(* CODESYS project PackML_Example_RECOVERED_2024-11-19T12-11-37.project
   Title: PackML Example
   Version: 1.0.0.0
   Author: 3S - Smart Software Solutions GmbH
   Description: Example project for the PackML State Machine library.
   Company: 3S - Smart Software Solutions GmbH

Project tree, tasks and I/O mapping:
  Device : CODESYS Control Win V3 x64, CODESYS, version 3.5.20.0
    application PackMLUnitModeManager
      libraries: OMAC PackML State Machine, 1.0.0.4 (3S - Smart Software Solutions GmbH); Standard, 3.5.18.0 (System)
      task MainTask (cyclic, interval t#20ms, priority 1) calls PLC_PRG
      task VISU_TASK (cyclic, interval 100 ms, priority 31) calls VisuElems.Visu_Prg
      global variables GVL
      program PLC_PRG [ST]: SimulateActingStateComplete
      visualisation Visualization
    SoftMotion General Axis Pool : SoftMotion General Axis Pool, CODESYS, version 4.11.0.0
      Axis : SM_Drive_Virtual, 3S - Smart Software Solutions GmbH, order no. 1805, version 4.0.0.0
          settings: wDriveID = 3; iMovementType = 0; fSWMaxVelocity = 1e3; fSWMaxAcceleration = 1e5; fSWMaxDeceleration = 1e5
  Device2 : CODESYS Control Win V3 x64, CODESYS, version 3.5.20.0
    application PackMLAxisControl
      libraries: OMAC PackML State Machine, 1.0.0.4 (3S - Smart Software Solutions GmbH)
      task Task (cyclic, interval t#20ms, priority 1) calls PLC_PRG
      task VISU_TASK (cyclic, interval 100 ms, priority 31) calls VisuElems.Visu_Prg
      program PLC_PRG [ST]
      function block AxisControl [ST]
      image pool ImagePool
      visualisation Visualization
    SoftMotion General Axis Pool : SoftMotion General Axis Pool, CODESYS, version 4.11.0.0
      Axis : SM_Drive_Virtual, 3S - Smart Software Solutions GmbH, order no. 1805, version 4.0.0.0
          settings: wDriveID = 2; iMovementType = 0; fSWMaxVelocity = 1e3; fSWMaxAcceleration = 1e5; fSWMaxDeceleration = 1e5
  MyPackML : CODESYS Control Win V3 x64, CODESYS, version 3.5.20.0
    application Application
      libraries: OMAC PackML State Machine, 1.0.0.4 (3S - Smart Software Solutions GmbH); Standard, 3.5.18.0 (System)
      PackML/
        function block MyUnitMode [ST]
        function block FB_Generic [ST]: M_Clearing, M_Init, M_Complete, M_Suspended, ParseStateToString, M_Idle, M_Log, M_Held, M_Aborted, GenerateErrorMsg, M_Completing, M_Execute, M_Stopped, Callback, M_Unsuspending, M_Starting, M_Holding, M_Suspending, M_CheckError, M_Resetting, M_StateComplete, M_Aborting, M_Stopping, M_Unholding, M_mapping, M_Undefined
        PackML/
          State and Mode/
            data type E_PMLProtectedUnitMode
            data type ST_PMLSubUnitInfo
            data type E_PMLCommand
            data type E_PMLState
          data type ST_PMLStateMachineOptions
          global variables G_PML
          data type ST_PMLUnitModeConfiguration
          data type ST_ChangeIntoProduction
          ITFs/
            interface I_UnitState: M_Idle, M_Holding, M_Unholding, M_Stopped, M_Execute, M_Held, M_Starting, M_Complete, M_Aborted, M_Suspended, M_Clearing, M_Stopping, M_Reseting, M_StateComplete, M_Aborting, M_Undefined, M_Unsuspending, M_Suspending, M_Completing
            interface I_UnitStateActing: M_Unholding, M_Execute, M_Completing, M_Reseting, M_Starting, M_Holding, M_Suspending, M_Unsuspending, M_Clearing, M_StateComplete, M_Aborting, M_Stopping
            interface I_UnitStateWaiting: M_Held, M_Idle, M_Undefined, M_Stopped, M_Suspended, M_Aborted, M_Complete
          data type ST_PMLSubUnitInfoRef
          Machine State/
            function block PML_UnitModeConfig [ST]
            function block PML_StateMachine [ST]: _supportedStates, M_NextState, M_StateComplete
            function block PML_UnitModeManager [ST]: M_SwitchUnitMode, M_Register
          PackTags/
            data type ST_PackMLv30
            Common/
              data type ST_Product
              data type ST_Interface
              data type ST_Descriptor
              data type ST_EquipmentInterlock
              data type ST_Ingredient
              data type ST_Alarm
              data type ST_Count
            data type ST_PMLs
            data type ST_PMLc
            data type ST_PMLa
        PubSub/
          interface I_SubCallback: Callback
          interface I_PubSubService: Unsubscribe, Subscribe, Publish
          data type E_Topics
          data type PubSubData
          global variables G_PubSub
          function block PubSubService [ST]: Publish, Subscribe, Unsubscribe
          data type SubscriberCell
          data type KeyAndValue
        image pool ImagePool
        function block FB_Machine [ST]: M_Clearing, M_Starting, M_SetUnitInfo, M_Resetting
        function block FB_Sample [ST]: Callback, M_Completing, M_Resetting, ParseStateToString, M_Stopping, M_Holding, M_Starting, M_agingTest, M_Execute, M_Undefined, M_Idle, M_mapping, M_Aborting, M_Reset
        function block MyUnitModeManager [ST]
        DUTs/
          data type E_UnitName
          interface I_Common: M_Init, ParseStateToString, GenerateErrorMsg, M_Log
          data type ST_UnitInfo
          data type E_SampleStates
          data type E_PMLSupportState
          data type E_PMLUserUnitMode
          data type E_ServerityLevelType
        global variables GVL
  libraries: VisuSymbols, 4.5.0.0 (System)
  5ce3da45-db07-42e7-a21c-a00fff4ed8f6|C:\Users\a.werner\Documents\background.jpg
  5ce3da45-db07-42e7-a21c-a00fff4ed8f6|C:\Users\a.werner\Documents\background.jpg
  text list GlobalTextList
*)

// MyPackML/Application/PackML/PackML/State and Mode/E_PMLProtectedUnitMode
{attribute 'qualified_only'}
{attribute 'strict'}
TYPE E_PMLProtectedUnitMode :
(
	ePMLProtUnitMode_Invalid		:=	0,
	ePMLProtUnitMode_Production		:=	1,
	ePMLProtUnitMode_Maintenance	:= 	2,
	ePMLProtUnitMode_Manual	 		:=	3
);
END_TYPE

// MyPackML/Application/PackML/PackML/PackTags/ST_PackMLv30
TYPE ST_PackMLv30 :
STRUCT
	Command	: ST_PMLc;
	Status	: ST_PMLs;
	Admin	: ST_PMLa;
END_STRUCT
END_TYPE

// MyPackML/Application/PackML/PackML/ST_PMLStateMachineOptions
TYPE ST_PMLStateMachineOptions :
STRUCT
END_STRUCT
END_TYPE

// MyPackML/Application/PackML/PackML/PackTags/Common/ST_Product
TYPE ST_Product :
STRUCT
	 /// 
	 ///Product identification number 
	 ProductID: DINT; 
	 /// 
	 ///Parameters required for processing given product 
	 ProcessVariables: ARRAY[1..G_PML.MaxProductProcessVariables] OF ST_Descriptor; 
	 /// 
	 ///Ingredients required for processing given product 
	 Ingredients: ARRAY[1..G_PML.MaxIngredients] OF ST_Ingredient;	
END_STRUCT
END_TYPE

// MyPackML/Application/PackML/PackML/ST_PMLUnitModeConfiguration
TYPE ST_PMLUnitModeConfiguration :
	STRUCT
		bActive				: BOOL;				
		aStateDisabled		: ARRAY [E_PMLState.ePMLState_Undefined..E_PMLState.ePMLState_Complete] OF BOOL;				
		aModeChangeValid	: ARRAY [E_PMLState.ePMLState_Undefined..E_PMLState.ePMLState_Complete] OF BOOL;			
		sName				: STRING;
	END_STRUCT	
END_TYPE

// MyPackML/Application/PackML/PackML/ST_ChangeIntoProduction
//structure for a visu userwindow, to chnage into productionmode
TYPE ST_ChangeIntoProduction :
STRUCT
	bYes		: BOOL;
	bNo			: BOOL;
	bYesReset	: BOOL;
END_STRUCT
END_TYPE

// MyPackML/Application/PackML/DUTs/E_UnitName
//Enumeration for Machineunits
TYPE E_UnitName :
(
	eMachine		:= 1,
	eSample			:= 2
				
)DINT;
END_TYPE

// MyPackML/Application/PackML/PackML/PackTags/Common/ST_Interface
TYPE ST_Interface :
STRUCT
	 /// 
	 ///Identification number of upstream or downstream unit machine 
	 Number: DINT; 
	 /// 
	 ///Control command for upstream or downstream machine 
	 ControlCmdNumber: DINT; 
	 /// 
	 ///Control command value associated with ControlCmdNumber 
	 CmdValue: DINT; 
	 /// 
	 ///Parameter data required for peer-to-peer coordination 
	 Parameter: ARRAY[1..G_PML.MaxInterfaceParameters] OF ST_Descriptor;
END_STRUCT
END_TYPE

// MyPackML/Application/PackML/PackML/PackTags/Common/ST_Descriptor
TYPE ST_Descriptor :
STRUCT
	 /// 
	 ///Parameter identification number 
	 ID: DINT; 
	 /// 
	 ///Parameter description 
	 Name: STRING; 
	 /// 
	 ///Parameter units of measure 
	 Unit: STRING; 
	 /// 
	 ///Numeric value of parameter 
	 Value: REAL;
END_STRUCT
END_TYPE

// MyPackML/Application/PackML/DUTs/ST_UnitInfo
//structure includes unit information
TYPE ST_UnitInfo :
STRUCT
	Name		: STRING;
	ActState	: E_PMLState;
	ActMode		: DINT;
END_STRUCT
END_TYPE

// MyPackML/Application/PackML/PackML/PackTags/ST_PMLs
TYPE ST_PMLs :
STRUCT
	/// 
	///Numeric representation of the active unit mode (required) 
	UnitModeCurrent: DINT; 
	/// 
	///Handshaking bit acknowledging that unit mode change request has been made. 
	UnitModeRequested: BOOL; 
	/// 
	///Signals that unit mode change request has been accepted; switching is actively in process. 
	UnitModeChangeInProcess: BOOL; 
	/// 
	///Numeric representation of the active state (required) 
	StateCurrent: DINT; 
	/// 
	///Handshaking value acknowledging that state change request has been made. 
	StateRequested: DINT; 
	/// 
	///Signals that state change request has been accepted; switching is actively in process. 
	StateChangeInProcess: BOOL; 
	/// 
	///Active machine speed setpoint in units of [primary packages/min] (required) 
	MachSpeed: REAL; 
	/// 
	///Actual machine speed in units of [primary packages/min] (required) 
	CurMachSpeed: REAL; 
	/// 
	///Bitwise indication that materials are ready for processing. 
	MaterialInterlock: ARRAY[0..31] OF BOOL; 
	/// 
	///Signals that the machine is either blocked or starved (required) 
	EquipmentInterlock: ST_EquipmentInterlock; 
	/// 
	///Use to coordinate activities between peers (i.e. upstream or downstream unit machines.) 
	RemoteInterface: ARRAY [1..G_PML.MaxStatusRemoteInterfaces] OF ST_Interface; 
	/// 
	///Current values or parameters associated to the end user supervisory interface. 
	Parameter: ARRAY [1..G_PML.MaxStatusParameters] OF ST_Descriptor; 
	/// 
	///Current recipe or process data associated to the various products run on the unit machine. 
	Product: ARRAY [1..G_PML.MaxStatusProducts] OF ST_Product;	
END_STRUCT
END_TYPE

// MyPackML/Application/PackML/DUTs/E_SampleStates
{attribute 'qualified_only'}
{attribute 'strict'}
TYPE E_SampleStates :
(
	IDLE := 0,
	INIT,
	CHECK,
	WAIT,
	WAIT_ON,
	WAIT_OFF,
	DETECTION,
	LAMP_ON,
	LAMP_OFF,
	DONE,

	ERROR
);
END_TYPE

// MyPackML/Application/PackML/PackML/State and Mode/ST_PMLSubUnitInfo
TYPE ST_PMLSubUnitInfo :
STRUCT
	Active	: BOOL;				
	eState	: E_PMLState	:=	E_PMLState.ePMLState_Aborted;	
END_STRUCT
END_TYPE

// MyPackML/Application/PackML/PackML/PackTags/ST_PMLc
TYPE ST_PMLc :
STRUCT
	/// 
	///Numeric representation of the commanded unit mode (required) 
	UnitMode: DINT; 
	/// 
	///Signals request that the current value of Command.UnitMode be activated (required) 
	UnitModeChangeRequest: BOOL; 
	/// 
	///Machine speed setpoint in units of [primary packages/min] (required) 
	MachSpeed: REAL; 
	/// 
	///Bitwise indication that materials are ready for processing. 
	MaterialInterlock: ARRAY[1..32] OF BOOL; 
	/// 
	///Numerical representation of the state commands (1=Reset, 2=Start, etc.) (required) 
	CntrlCmd: DINT; 
	/// 
	///Signals request that the current value of Command.CntrlCmd be activated (required) 
	CmdChangeRequest: BOOL; 
	///
	///Use to coordinate activities between peers (i.e. upstream or downstream unit machines.) 
	RemoteInterface: ARRAY [1..G_PML.MaxCommandRemoteInterfaces] OF ST_Interface; 
	/// 
	///Values or parameters associated to the end user supervisory interface. 
	Parameter: ARRAY [1..G_PML.MaxCommandParameters] OF ST_Descriptor; 
	/// 
	///Recipe or process data associated to the various products run on the unit machine. 
	Product: ARRAY [1..G_PML.MaxCommandProducts] OF ST_Product;
	
END_STRUCT
END_TYPE

// MyPackML/Application/PackML/PubSub/E_Topics
TYPE E_Topics :
(
	UNKNOWN 				:= 0, 
	SAMPLE_SUBSCRRIBE_1		:= 1, 
	SAMPLE_SUBSCRRIBE_2		:= 2, 
	SAMPLE_SUBSCRRIBE_3		:= 3,
	NUMBER_OF_TOPICS
);
END_TYPE

// MyPackML/Application/PackML/PackML/ST_PMLSubUnitInfoRef
TYPE ST_PMLSubUnitInfoRef :
STRUCT
	//pArray			: PVOID;//codesys don't have pvoid yet	
	pArray			: POINTER TO ST_PMLSubUnitInfo;		
	ArraySize		: UDINT;				
	NoOfSubUnits	: UDINT;	
END_STRUCT
END_TYPE

// MyPackML/Application/PackML/PackML/PackTags/Common/ST_EquipmentInterlock
TYPE ST_EquipmentInterlock :
STRUCT
	/// 
	///Machine stoppage due to downstream fault 
	Blocked: BOOL; 
	/// 
	///Machine stoppage due to upstream or supply fault 
	Starved: BOOL;
END_STRUCT
END_TYPE

// MyPackML/Application/PackML/PubSub/PubSubData
TYPE PubSubData :
STRUCT
	Topic : E_Topics;
	Data	: ARRAY[0..MAX_PUB_SUB_DATA] OF KeyAndValue;
END_STRUCT
END_TYPE

// MyPackML/Application/PackML/PackML/PackTags/Common/ST_Ingredient
TYPE ST_Ingredient: 
STRUCT 
	 /// 
	 ///Ingredient identification number 
	 IngredientID: DINT; 
	 /// 
	 ///Parameters associated to given ingredient 
	 Parameter: ARRAY[1..G_PML.MaxIngredientParameters] OF ST_Descriptor; 
END_STRUCT 
END_TYPE

// MyPackML/Application/PackML/DUTs/E_PMLSupportState
{attribute 'qualified_only'}
{attribute 'strict'}
TYPE E_PMLSupportState :
(
	Stopped := 16#1, // Bit 0
	Resetting := 16#2, // Bit 1
	Idle := 16#4, // Bit 2
	Starting := 16#8, // Bit 3
	Execute := 16#10, // Bit 4
	Holding := 16#20, // Bit 5
	Held := 16#40, // Bit 6
	UnHolding := 16#80, // Bit 7
	Suspending := 16#100, // Bit 8
	Suspended := 16#200, // Bit 9
	UnSuspending := 16#400, // Bit 10
	Completing := 16#800, // Bit 11
	Complete := 16#1000, // Bit 12
	Stopping := 16#2000, // Bit 13
	Aborting := 16#4000, // Bit 14
	Aborted := 16#8000, // Bit 15
	Clearing := 16#10000, // Bit 16
	
	No := 0,
	All := 16#1FFFF,
	Invalid := 16#80000000
) DWORD;
END_TYPE

// MyPackML/Application/PackML/PackML/State and Mode/E_PMLCommand
{attribute 'strict'}
TYPE E_PMLCommand :
(
	ePMLCommand_Undefined		:=	0,	
	ePMLCommand_Reset			:=	1,	
	ePMLCommand_Start			:=	2,	
	ePMLCommand_Stop			:=	3,	
	ePMLCommand_Hold			:=	4,	
	ePMLCommand_Unhold			:=	5,	
	ePMLCommand_Suspend			:=	6,	
	ePMLCommand_Unsuspend		:=	7,	
	ePMLCommand_Abort			:=	8,	
	ePMLCommand_Clear			:=	9,	
	//	extension TO OMAC TR88.00.02
	ePMLCommand_Complete		:=	10
);
END_TYPE

// MyPackML/Application/PackML/PackML/PackTags/Common/ST_Alarm
TYPE ST_Alarm: 
STRUCT 
	 /// 
	 ///Alarm or warning current status 
	 Trigger: BOOL; 
	 /// 
	 ///Alarm or warning identification number 
	 ID: DINT; 
	 /// 
	 ///Context specific value associated to given alarm or warning 
	 Value: DINT; 
	 /// 
	 ///Alarm or warning description 
	 Message: STRING; 
	 /// 
	 ///Identification number associated to alarm type or severity 
	 Category: DINT; 
	 /// 
	 ///Time stamp of alarm or warning occurrence. Format year:month:day:hour:min:sec:µsec 
	 DateTime: ARRAY[0..6] OF DINT; 
	 /// 
	 ///Time stamp of alarm or warning acknowledgment. Format year:month:day:hour:min:sec:µsec 
	 AckDateTime: ARRAY[0..6] OF DINT; 
END_STRUCT 
END_TYPE

// MyPackML/Application/PackML/PackML/PackTags/Common/ST_Count
TYPE ST_Count :
STRUCT
	 /// 
	 ///Product identification number 
	 ID: DINT; 
	 /// 
	 ///Product description 
	 Name: STRING; 
	 /// 
	 ///Product unit of measure 
	 Unit: STRING; 
	 /// 
	 ///Count since last operator reset 
	 Count: DINT; 
	 /// 
	 ///Count since last accumulative counter reset 
	 AccCount: DINT;
END_STRUCT
END_TYPE

// MyPackML/Application/PackML/DUTs/E_PMLUserUnitMode
//Enumeration for User Modes
TYPE E_PMLUserUnitMode : (
	ePMLUnitMode_Service		:=  4,
	ePMLUnitMode_Usermode2		:=  5,
	ePMLUnitMode_Usermode3		:=  6,
	ePMLUnitMode_Usermode4		:=  7,
	ePMLUnitMode_Usermode5 		:=  8,
	ePMLUnitMode_Usermode6 		:=  9,
	ePMLUnitMode_Usermode7 		:=  10
) DINT;
END_TYPE

// MyPackML/Application/PackML/PubSub/SubscriberCell
TYPE SubscriberCell :
STRUCT
	occupied : BOOL;
	subscriber : I_SubCallback;
END_STRUCT
END_TYPE

// MyPackML/Application/PackML/PubSub/KeyAndValue
TYPE KeyAndValue :
STRUCT
	Key : STRING;
	Value : string;
END_STRUCT
END_TYPE

// MyPackML/Application/PackML/DUTs/E_ServerityLevelType
{attribute 'qualified_only'}
{attribute 'strict'}
TYPE E_ServerityLevelType :
(
	SERVICE := 0,
	ERROR,
	WARNING,
	INFO,
	DEBUG
);
END_TYPE

// MyPackML/Application/PackML/PackML/PackTags/ST_PMLa
TYPE ST_PMLa :
STRUCT
	/// 
	///Parameters associated to the local interface (e.g. HMI) 
	Parameter: ARRAY [1..G_PML.MaxAdminParameters] OF ST_Descriptor; 
	/// 
	///Listing of all currently active alarms 
	Alarm: ARRAY [1..G_PML.MaxAlarms] OF ST_Alarm; 
	/// 
	///Extent of the Alarm array 
	AlarmExtent: DINT	:= G_PML.MaxAlarms; 
	/// 
	///Chronological alarm history, with most recent given as AlarmHistory[0] 
	AlarmHistory: ARRAY [1..G_PML.MaxHistoryAlarms] OF ST_Alarm; 
	/// 
	///Extent of AlarmHistory array 
	AlarmHistoryExtent: DINT	:= G_PML.MaxHistoryAlarms; 
	/// 
	///Alarm associated to the primary cause of machine stoppage ('first fault') (required) 
	StopReason: ARRAY [1..G_PML.MaxStopReasons] OF ST_Alarm; 
	/// 
	///Extent of StopReason array 
	StopReasonExtent: DINT	:= G_PML.MaxStopReasons; 
	/// 
	///Listing of all currently active warnings 
	Warning: ARRAY [1..G_PML.MaxWarnings] OF ST_Alarm; 
	/// 
	///Extent of warning array 
	WarningExtent: DINT	:= G_PML.MaxWarnings; 
	/// 
	///Elapsed time in seconds of current mode. 
	ModeCurrentTime: ARRAY [0..G_PML.MaxUnitMode] OF DINT;
	/// 
	///Cumulative time in seconds in each defined mode. 
	ModeCumulativeTime: ARRAY [0..G_PML.MaxUnitMode] OF DINT; 
	/// 
	///Elapsed time in seconds of current [mode, state] pair. 
	StateCurrentTime: ARRAY [0..G_PML.MaxUnitMode, 0..G_PML.MaxMachineState] OF DINT; 
	/// 
	///Cumulative time in seconds in each defined [mode, state] pair. 
	StateCumulativeTime: ARRAY [0..G_PML.MaxUnitMode, 0..G_PML.MaxMachineState] OF DINT; 
	/// 
	///Count of raw materials used or consumed during production 
	ProdConsumedCount: ARRAY [1..G_PML.MaxConsumedCounts] OF ST_Count; 
	/// 
	///Count of total products (i.e. good + defective) made during production (required) 
	ProdProcessedCount: ARRAY [1..G_PML.MaxProductCounts] OF ST_Count; 
	/// 
 	///Count of defective products made during production. (required) 
	ProdDefectiveCount: ARRAY [1..G_PML.MaxProductCounts] OF ST_Count; 
	/// 
	///Accumulative time since last reset of timer arrays. 
	AccTimeSinceReset: DINT; 	
	/// 
	///Maximum design speed of the machine within given environment. 
	MachDesignSpeed: REAL; 	
	/// 
	///Bitwise indication of inactive states in current mode. 
	StatesDisabled: DINT; 		
	/// 
	///Current date and time of local processing unit (PLC, PC, PAC, microcontroller, etc.) 
	PLCDateTime: ARRAY[0..6] OF DINT;
END_STRUCT
END_TYPE

// MyPackML/Application/PackML/PackML/State and Mode/E_PMLState
TYPE E_PMLState :
(
	//states according TO PackTags v3.0
	ePMLState_Undefined		:=			0,	
	ePMLState_Clearing		:=			1,	
	ePMLState_Stopped		:=			2,	
	ePMLState_Starting		:=			3,	
	ePMLState_Idle			:=			4,	
	ePMLState_Suspended		:=			5,	
	ePMLState_Execute		:=			6,	
	ePMLState_Stopping		:=			7,	
	ePMLState_Aborting		:=			8,	
	ePMLState_Aborted		:=			9,	
	ePMLState_Holding		:=			10,	
	ePMLState_Held			:=			11,	
	ePMLState_Unholding		:=			12,	
	ePMLState_Suspending	:=			13,	
	ePMLState_Unsuspending	:=			14,	
	ePMLState_Resetting		:=			15,	
	ePMLState_Completing	:=			16,	
	ePMLState_Complete		:=			17
);
END_TYPE

// MyPackML/Application/PackML/PackML/G_PML
{attribute 'qualified_only'}
VAR_GLOBAL CONSTANT
	MaxInterfaceParameters		: INT	:=5;	//PMLc/PMLs
	MaxProductProcessVariables	: INT	:=10;
	MaxIngredients				: INT	:=10;
	MaxIngredientParameters		: INT	:=10;
	MaxCommandRemoteInterfaces	: INT	:=2;	//PMLc
	MaxCommandParameters		: INT	:=10;	
	MaxCommandProducts			: INT	:=5;
	MaxStatusRemoteInterfaces	: INT	:=2;	//PMLs
	MaxStatusParameters			: INT	:=10;	
	MaxStatusProducts			: INT	:=5;	
	MaxAdminParameters			: INT	:=10;	//PMLa
	MaxAlarms					: INT	:=10;	
	MaxHistoryAlarms			: INT	:=10;	
	MaxStopReasons				: INT	:=10;	
	MaxWarnings					: INT	:=10;	
	MaxConsumedCounts			: INT	:=10;	
	MaxProductCounts			: INT	:=10;
	
	MaxUnitMode					:INT	:=31;
	MaxMachineState				:INT	:=17;
	stPMLUnitModeConfiguration	:ARRAY [0..MaxUnitMode] OF ST_PMLUnitModeConfiguration	:=	[STRUCT(bActive := TRUE, sName := 'Invalid', aStateDisabled := [18(FALSE)], aModeChangeValid := [18(TRUE)]), 
																							 STRUCT(bActive := TRUE, sName := 'Production', aStateDisabled := [18(FALSE)], aModeChangeValid := [TRUE, FALSE, TRUE, FALSE, TRUE, FALSE, FALSE, FALSE, FALSE, TRUE, FALSE, TRUE, FALSE, FALSE, FALSE, FALSE, FALSE, FALSE]), 
																							 STRUCT(bActive := TRUE, sName := 'Maintenance', aStateDisabled := [FALSE, FALSE, FALSE, FALSE, FALSE, TRUE, FALSE, FALSE, FALSE, FALSE, FALSE, FALSE, FALSE, TRUE, TRUE, FALSE, TRUE, TRUE], aModeChangeValid := [TRUE, FALSE, TRUE, FALSE, TRUE, FALSE, FALSE, FALSE, FALSE, TRUE, FALSE, TRUE, FALSE, FALSE, FALSE, FALSE, FALSE, FALSE]), 
																							 STRUCT(bActive := TRUE, sName := 'Manual', aStateDisabled := [FALSE, FALSE, FALSE, FALSE, FALSE, TRUE, FALSE, FALSE, FALSE, FALSE, TRUE, TRUE, TRUE, TRUE, TRUE, FALSE, TRUE, TRUE], aModeChangeValid := [TRUE, FALSE, TRUE, FALSE, TRUE, FALSE, FALSE, FALSE, FALSE, TRUE, FALSE, FALSE, FALSE, FALSE, FALSE, FALSE, FALSE, FALSE])];	
END_VAR

// Device/PackMLUnitModeManager/GVL
VAR_GLOBAL CONSTANT
	gc_sPRODUCTION 	: STRING := 'Production';
	gc_sSEMIAUTO 	: STRING := 'Semi Auto';
	gc_sSETUP 		: STRING := 'Setup';
	gc_sUSER		: STRING := 'User';
END_VAR

// MyPackML/Application/PackML/PubSub/G_PubSub

VAR_GLOBAL CONSTANT
	MAX_PUB_SUB_DATA	: INT:=19;
END_VAR

// MyPackML/Application/PackML/GVL
VAR_GLOBAL CONSTANT
	gc_sPRODUCTION : STRING := 'Production';
	gc_sSEMIAUTO : STRING := 'Semi Auto';
	gc_sSETUP : STRING := 'Setup';
END_VAR
{attribute 'qualified_only'}
VAR_GLOBAL
	packTags	: ST_PackMLv30;
	bButtonProductionReq		: BOOL;							//TRUE when a mode change to PRODUCTION is requested
	stChangeIntoProduction		: ST_ChangeIntoProduction;		//Result of command box "Change to Production requested"
	
	PubSubService	: PubSubService;

	pml_adminAlarm	: PML_AdminAlarm;
	
	aUnitInfo					: ARRAY [1..12] OF ST_UnitInfo;	//Array includes the states and modes of machineunits	
	aCaption					: ARRAY [1..12] OF STRING := ['F1','F2','F3','F4','F5','F6','F7','F8','F9','F10','F11','F12'];
	aKeyPressed					: ARRAY [1..12] OF BOOL;


	fb_sample	: FB_Sample;		
END_VAR

// Device2/PackMLAxisControl/PLC_PRG
PROGRAM PLC_PRG
VAR
	xInit				: BOOL := FALSE; // Flag for initialization

	ac: AxisControl;
	
	// Visu Commands	
	xAbort				: BOOL;
	xActingStateComplete: BOOL;
	xClear				: BOOL;
	xHold				: BOOL;
	xReset				: BOOL;
	xStart				: BOOL;
	xStop				: BOOL;
	xSuspend			: BOOL;
	xUnHold				: BOOL;
	xUnSuspend			: BOOL;
	
	
END_VAR

ac(Axis:=Axis);

// Visu commands
IF xAbort THEN
	ac.ItfUnitMode.Abort();
END_IF
IF xClear THEN
	ac.ItfUnitMode.Clear();
END_IF
IF xHold THEN
	ac.ItfUnitMode.Hold();
END_IF
IF xReset THEN
	ac.ItfUnitMode.Reset();
END_IF
IF xStart THEN
	ac.ItfUnitMode.Start();
END_IF
IF xStop THEN
	ac.ItfUnitMode.Stop();
END_IF
IF xSuspend THEN
	ac.ItfUnitMode.Suspend();
END_IF
IF xUnHold THEN
	ac.ItfUnitMode.UnHold();
END_IF
IF xUnSuspend THEN
	ac.ItfUnitMode.UnSuspend();
END_IF
IF xActingStateComplete AND ac.ItfUnitMode.CurrentState = PACK_ML.State.Execute THEN
	ac.ItfUnitMode.ActingStateCompleted();
END_IF

END_PROGRAM

// Device/PackMLUnitModeManager/PLC_PRG
// Example project for the PackML State Machine with three unit modes.
PROGRAM PLC_PRG
VAR
	productionUnitMode	: PACK_ML.UnitMode; // Example unit mode for prodction
	semiAutoUnitMode	: PACK_ML.UnitMode; // Example unit mode for semi auto production
	setupUnitMode		: PACK_ML.UnitMode; // Example unit mode for setup
	userUnitMode		: PACK_ML.UnitMode; // Example unit mode for setup
	unitModeManager		: PACK_ML.UnitModeManager; // Unit mode manager to switch between unitmodes
	currentUnitMode		: PACK_ML.IUnitMode;
	xInit				: BOOL := FALSE; // Flag for initialization
	
	// Visu Commands	
	xAbort				: BOOL;
	xActingStateComplete: BOOL;
	xClear				: BOOL;
	xHold				: BOOL;
	xReset				: BOOL;
	xStart				: BOOL;
	xStop				: BOOL;
	xSuspend			: BOOL;
	xUnHold				: BOOL;
	xUnSuspend			: BOOL;
	
	// Helper
	xSimulate			: BOOL;
	xChangeState		: BOOL := FALSE;	
	timer1				: TON;	
	iSelectedUnitMode	: INT := 0;
	iLastSelectedUnitMode: INT := 0;
	xUserModeChanged	: BOOL;
	
END_VAR

IF NOT xInit THEN
	productionUnitMode(		sName := gc_sPRODUCTION, 
							dwSupportedStates := PACK_ML.State.All, 
							dwAllowsLeavingFromStates := PACK_ML.State.Stopped OR PACK_ML.State.Aborted OR PACK_ML.State.Idle, 
							dwAllowsEnteringIntoStates := PACK_ML.State.Stopped OR PACK_ML.State.Aborted OR PACK_ML.State.Idle, 
							eInitialState := PACK_ML.State.Idle,
							xActive := TRUE);
	semiAutoUnitMode(		sName := gc_sSEMIAUTO, 
							dwSupportedStates := PACK_ML.State.All - PACK_ML.State.Completing - PACK_ML.State.Complete - PACK_ML.State.Holding - PACK_ML.State.Held - PACK_ML.State.UnHolding,
							dwAllowsLeavingFromStates := PACK_ML.State.Stopped OR PACK_ML.State.Aborted OR PACK_ML.State.Idle, 
							dwAllowsEnteringIntoStates := PACK_ML.State.Stopped OR PACK_ML.State.Aborted OR PACK_ML.State.Idle,   
							eInitialState := PACK_ML.State.Idle, 
							xActive := FALSE);
	setupUnitMode(			sName := gc_sSETUP, 
							dwSupportedStates := PACK_ML.State.All - PACK_ML.State.Completing - PACK_ML.State.Complete - PACK_ML.State.Holding - PACK_ML.State.Held - PACK_ML.State.UnHolding - PACK_ML.State.UnSuspending - PACK_ML.State.Suspended - PACK_ML.State.Suspending,
							dwAllowsLeavingFromStates := PACK_ML.State.Stopped OR PACK_ML.State.Aborted OR PACK_ML.State.Idle,   
							dwAllowsEnteringIntoStates := PACK_ML.State.Stopped OR PACK_ML.State.Aborted OR PACK_ML.State.Idle, 
							eInitialState := PACK_ML.State.Idle, 
							xActive := FALSE);
	userUnitMode(			sName := gc_sUSER, 
							dwSupportedStates := PACK_ML.State.All - PACK_ML.State.Completing - PACK_ML.State.Complete - PACK_ML.State.Holding - PACK_ML.State.Held - PACK_ML.State.UnHolding - PACK_ML.State.UnSuspending - PACK_ML.State.Suspended - PACK_ML.State.Suspending-PACK_ML.State.Clearing-PACK_ML.Aborted,
							dwAllowsLeavingFromStates := PACK_ML.State.Stopped OR PACK_ML.State.Aborted OR PACK_ML.State.Idle,   
							dwAllowsEnteringIntoStates := PACK_ML.State.Stopped OR PACK_ML.State.Aborted OR PACK_ML.State.Idle, 
							eInitialState := PACK_ML.State.Idle, 
							xActive := FALSE);
	// Register the unit modes 
	unitModeManager.Register(productionUnitMode);
	unitModeManager.Register(semiAutoUnitMode);
	unitModeManager.Register(setupUnitMode);
	unitModeManager.Register(userUnitMode);
	xInit := TRUE;
END_IF

IF unitModeManager.ActiveUnitMode <> 0 THEN	
	currentUnitMode := unitModeManager.ActiveUnitMode;
	
	// Visu commands
	IF xAbort THEN
		unitModeManager.ActiveUnitMode.Abort();
	END_IF
	IF xClear THEN
		unitModeManager.ActiveUnitMode.Clear();
	END_IF
	IF xHold THEN
		unitModeManager.ActiveUnitMode.Hold();
	END_IF
	IF xReset THEN
		unitModeManager.ActiveUnitMode.Reset();
	END_IF
	IF xStart THEN
		unitModeManager.ActiveUnitMode.Start();
	END_IF
	IF xStop THEN
		unitModeManager.ActiveUnitMode.Stop();
	END_IF
	IF xSuspend THEN
		unitModeManager.ActiveUnitMode.Suspend();
	END_IF
	IF xUnHold THEN
		unitModeManager.ActiveUnitMode.UnHold();
	END_IF
	IF xUnSuspend THEN
		unitModeManager.ActiveUnitMode.UnSuspend();
	END_IF
	IF xActingStateComplete AND NOT xSimulate THEN
		unitModeManager.ActiveUnitMode.ActingStateCompleted();
	END_IF
	
	// Simulate action complete
	SimulateActingStateComplete();	 
END_IF

// Change the current unit mode
IF iSelectedUnitMode <> iLastSelectedUnitMode THEN
	CASE iSelectedUnitMode OF 
		0:
			xUserModeChanged := unitModeManager.SwitchUnitMode(gc_sPRODUCTION);
		1:
			xUserModeChanged := unitModeManager.SwitchUnitMode(gc_sSEMIAUTO);
		2:
			xUserModeChanged := unitModeManager.SwitchUnitMode(gc_sSETUP);
		3:
			xUserModeChanged := unitModeManager.SwitchUnitMode(gc_sUser);
	END_CASE
	IF xUserModeChanged THEN
		iLastSelectedUnitMode := iSelectedUnitMode;
	ELSE
		iSelectedUnitMode := iLastSelectedUnitMode;
	END_IF
END_IF

METHOD SimulateActingStateComplete
VAR_INPUT
END_VAR
VAR
	nextSupportedState	: UDINT;	
END_VAR
nextSupportedState := unitModeManager.ActiveUnitMode.NextState(unitModeManager.ActiveUnitMode.CurrentState);	
IF nextSupportedState = PACK_ML.State.Execute OR nextSupportedState = PACK_ML.State.Completing OR nextSupportedState = PACK_ML.State.Complete OR nextSupportedState = PACK_ML.State.Held OR nextSupportedState = PACK_ML.State.Aborted OR nextSupportedState = PACK_ML.State.Stopped OR nextSupportedState = PACK_ML.State.Idle OR nextSupportedState = PACK_ML.State.Suspended THEN	
	timer1(IN := TRUE, PT := T#2S, Q => xChangeState);
	xSimulate := TRUE;
END_IF   
IF xChangeState THEN
	unitModeManager.ActiveUnitMode.ActingStateCompleted();
	timer1(IN := FALSE);
	xSimulate := FALSE;
	xChangeState := FALSE;
END_IF
END_METHOD

END_PROGRAM

// Device2/PackMLAxisControl/AxisControl
FUNCTION_BLOCK AxisControl
// This FB represents an axis, which is controlled according to its active unit mode
VAR_IN_OUT
	Axis: AXIS_REF_SM3;
END_VAR
VAR_OUTPUT
	ItfUnitMode	: PACK_ML.IUnitMode; // UnitMode of the axis
END_VAR
VAR
	UM	: PACK_ML.UnitMode; 

	xInit				: BOOL := FALSE; // Flag for initialization

	//motion FBs
	p: MC_Power;
	rs: MC_ReadStatus;
	res: MC_Reset;
	moverel: MC_MoveRelative;
	halt: MC_Halt;
	moveabs: MC_MoveAbsolute;
	h: MC_Home;
	
	
	tii	: TON;
END_VAR

IF NOT xInit THEN	
	UM				(		sName := 'Normal Operation', 
							dwSupportedStates := PACK_ML.State.All - PACK_ML.State.Suspending - PACK_ML.State.Suspended - PACK_ML.State.UnSuspending, 
							dwAllowsLeavingFromStates := PACK_ML.State.Stopped OR PACK_ML.State.Aborted OR PACK_ML.State.Idle, 
							dwAllowsEnteringIntoStates := PACK_ML.State.Stopped OR PACK_ML.State.Aborted OR PACK_ML.State.Idle, 
							eInitialState := PACK_ML.State.Aborted,
							xActive := TRUE);
	ItfUnitMode := UM; 
	xInit := TRUE;
END_IF

CASE UM.CurrentState OF
PACK_ML.State.Stopped,
PACK_ML.State.Aborted,
PACK_ML.State.Idle,
PACK_ML.State.Held,
PACK_ML.State.Complete :
	// in this waiting states we reset the Execute input of the moving FBs
	res.Execute := FALSE;
	moverel.Execute := FALSE;
	halt.Execute := FALSE;
	moveabs.Execute := FALSE;
	h.Execute := FALSE;
PACK_ML.State.Resetting :
	IF rs.Errorstop THEN	//first reset errors when necessary
		h.Execute := FALSE;
		IF res.Error THEN
			res.Execute := FALSE;
		ELSE	
			res.Execute := TRUE;
		END_IF
	ELSE
		p.bDriveStart := TRUE;	//release quickstop
		IF p.Status THEN
			h.Execute := TRUE;	//do homing
			IF h.Done THEN	
				h.Execute := FALSE;
				UM.ActingStateCompleted();
			END_IF
		END_IF
	END_IF
PACK_ML.State.Starting :
	moverel.Execute:=FALSE;
	UM.ActingStateCompleted();
PACK_ML.State.Execute :
	moverel.Execute:=TRUE;
	IF moverel.Done THEN
		moverel.Execute:=FALSE;
 	END_IF
PACK_ML.State.Holding :
	moverel.Execute:=FALSE;
	halt.Execute:=TRUE;
	IF halt.Done THEN
		halt.Execute := FALSE;
		UM.ActingStateCompleted();
	END_IF
PACK_ML.State.UnHolding :
	halt.Execute:=FALSE;
	moveabs.Execute := TRUE;
	IF moveabs.Done THEN
		moveabs.Execute := FALSE;
		UM.ActingStateCompleted();
	END_IF
PACK_ML.State.Completing :
	IF moverel.Done THEN
		UM.ActingStateCompleted();
	END_IF
PACK_ML.State.Aborting :
	p.bDriveStart := FALSE;
	p.bRegulatorOn := FALSE;
	UM.ActingStateCompleted();
PACK_ML.State.Stopping,
PACK_ML.State.Clearing :	
	p.bRegulatorOn:=TRUE; 
	p.bDriveStart:=FALSE; 
	IF p.bRegulatorRealState AND NOT p.bDriveStartRealState THEN
		UM.ActingStateCompleted();
	END_IF
END_CASE

p(
	Axis:=Axis , 
	Enable:=TRUE , 
	Status=> , 
	bRegulatorRealState=> , 
	bDriveStartRealState=> , 
	Busy=> , 
	Error=> , 
	ErrorID=> );

rs(
	Axis:=Axis , 
	Enable:=TRUE , 
	Valid=> , 
	Busy=> , 
	Error=> , 
	ErrorID=> , 
	Disabled=> , 
	Errorstop=> , 
	Stopping=> , 
	StandStill=> , 
	DiscreteMotion=> , 
	ContinuousMotion=> , 
	SynchronizedMotion=> , 
	Homing=> , 
	ConstantVelocity=> , 
	Accelerating=> , 
	Decelerating=> , 
	FBErrorOccured=> );
	
res(
	Axis:=Axis , 
	Execute:= , 
	Done=> , 
	Busy=> , 
	Error=> , 
	ErrorID=> );
	
moverel(
	Axis:=Axis , 
	Distance:=360 , 
	Velocity:=360 , 
	Acceleration:=360 , 
	Deceleration:=360, 
	Jerk:= , 
	Done=> , 
	Busy=> , 
	CommandAborted=> , 
	Error=> , 
	ErrorID=> );
	
moveabs(
	Axis:=Axis , 
	Execute:= , 
	Position:=0 , 
	Velocity:=360 , 
	Acceleration:=360 , 
	Deceleration:=360 , 
	Jerk:= , 
	Direction:=positive , 
	Done=> , 
	Busy=> , 
	CommandAborted=> , 
	Error=> , 
	ErrorID=> );
	
halt(
	Axis:=axis , 
	Execute:= , 
	Deceleration:=1000 , 
	Jerk:= , 
	Done=> , 
	Busy=> , 
	CommandAborted=> , 
	Error=> , 
	ErrorID=> );
	
h(
	Axis:=Axis , 
	Execute:= , 
	Position:= , 
	Done=> , 
	Busy=> , 
	CommandAborted=> , 
	Error=> , 
	ErrorID=> );

END_FUNCTION_BLOCK

// MyPackML/Application/PackML/PubSub/I_SubCallback
(*
Description: 
Interface that every function block that wants to be a subscriber, needs to implement.
*)
INTERFACE I_SubCallback

(*
Description: 
the callback that will be invoked when there is a publish for what the subscriber was subscribed to.
*)
METHOD Callback
VAR_INPUT
	data : PubSubData;
END_VAR
END_METHOD

END_INTERFACE

// MyPackML/Application/PackML/PackML/Machine State/PML_UnitModeConfig
//just to config the unit mode,can 
FUNCTION_BLOCK PML_UnitModeConfig
VAR_INPUT
	//
	eMode							: DINT;				
	sName							: STRING;
	//config which state disable				
	bDisableClearing				: BOOL;				
	bDisableStarting				: BOOL;				
	bDisableSuspended				: BOOL;				
	bDisableStopping				: BOOL;				
	bDisableAborting				: BOOL;				
	bDisableHolding					: BOOL;				
	bDisableHeld					: BOOL;				
	bDisableUnholding				: BOOL;				
	bDisableSuspending				: BOOL;				
	bDisableUnsuspending			: BOOL;				
	bDisableResetting				: BOOL;				
	bDisableIdle					: BOOL;				
	bDisableCompleting				: BOOL;				
	bDisableComplete				: BOOL;
	//config unit mode can be changed in which state				
	bEnableUnitModeChangeStopped	: BOOL;				
	bEnableUnitModeChangeIdle		: BOOL;				
	bEnableUnitModeChangeSuspended	: BOOL;				
	bEnableUnitModeChangeExecute	: BOOL;				
	bEnableUnitModeChangeAborted	: BOOL;				
	bEnableUnitModeChangeHeld		: BOOL;				
	bEnableUnitModeChangeComplete	: BOOL;		
END_VAR
VAR_OUTPUT
	bError	: BOOL;				
	nErrorId	: UDINT;	
END_VAR
VAR
END_VAR

END_FUNCTION_BLOCK

// MyPackML/Application/PackML/MyUnitMode
FUNCTION_BLOCK MyUnitMode
VAR_INPUT
END_VAR
VAR_OUTPUT
END_VAR
VAR
END_VAR

END_FUNCTION_BLOCK

// MyPackML/Application/PackML/PackML/ITFs/I_UnitState
INTERFACE I_UnitState EXTENDS I_UnitStateWaiting,I_UnitStateActing

METHOD M_Idle
VAR_INPUT
END_VAR
END_METHOD

METHOD M_Holding
VAR_INPUT
END_VAR
END_METHOD

METHOD M_Unholding
VAR_INPUT
END_VAR
END_METHOD

METHOD M_Stopped
VAR_INPUT
END_VAR
END_METHOD

METHOD M_Execute
VAR_INPUT
END_VAR
END_METHOD

METHOD M_Held
VAR_INPUT
END_VAR
END_METHOD

METHOD M_Starting
VAR_INPUT
END_VAR
END_METHOD

METHOD M_Complete
VAR_INPUT
END_VAR
END_METHOD

METHOD M_Aborted
VAR_INPUT
END_VAR
END_METHOD

METHOD M_Suspended
VAR_INPUT
END_VAR
END_METHOD

METHOD M_Clearing
VAR_INPUT
END_VAR
END_METHOD

METHOD M_Stopping
VAR_INPUT
END_VAR
END_METHOD

METHOD M_Reseting
VAR_INPUT
END_VAR
END_METHOD

METHOD M_StateComplete
VAR_INPUT
END_VAR
END_METHOD

METHOD M_Aborting
VAR_INPUT
END_VAR
END_METHOD

METHOD M_Undefined
VAR_INPUT
END_VAR
END_METHOD

METHOD M_Unsuspending
VAR_INPUT
END_VAR
END_METHOD

METHOD M_Suspending
VAR_INPUT
END_VAR
END_METHOD

METHOD M_Completing
VAR_INPUT
END_VAR
END_METHOD

END_INTERFACE

// MyPackML/Application/PackML/PackML/ITFs/I_UnitStateWaiting
INTERFACE I_UnitStateWaiting

METHOD M_Held
VAR_INPUT
END_VAR
END_METHOD

METHOD M_Idle
VAR_INPUT
END_VAR
END_METHOD

METHOD M_Undefined
VAR_INPUT
END_VAR
END_METHOD

METHOD M_Stopped
VAR_INPUT
END_VAR
END_METHOD

METHOD M_Suspended
VAR_INPUT
END_VAR
END_METHOD

METHOD M_Aborted
VAR_INPUT
END_VAR
END_METHOD

METHOD M_Complete
VAR_INPUT
END_VAR
END_METHOD

END_INTERFACE

// MyPackML/Application/PackML/PackML/ITFs/I_UnitStateActing
INTERFACE I_UnitStateActing

METHOD M_Unholding
VAR_INPUT
END_VAR
END_METHOD

METHOD M_Execute
VAR_INPUT
END_VAR
END_METHOD

METHOD M_Completing
VAR_INPUT
END_VAR
END_METHOD

METHOD M_Reseting
VAR_INPUT
END_VAR
END_METHOD

METHOD M_Starting
VAR_INPUT
END_VAR
END_METHOD

METHOD M_Holding
VAR_INPUT
END_VAR
END_METHOD

METHOD M_Suspending
VAR_INPUT
END_VAR
END_METHOD

METHOD M_Unsuspending
VAR_INPUT
END_VAR
END_METHOD

METHOD M_Clearing
VAR_INPUT
END_VAR
END_METHOD

METHOD M_StateComplete
VAR_INPUT
END_VAR
END_METHOD

METHOD M_Aborting
VAR_INPUT
END_VAR
END_METHOD

METHOD M_Stopping
VAR_INPUT
END_VAR
END_METHOD

END_INTERFACE

// MyPackML/Application/PackML/DUTs/I_Common
INTERFACE I_Common

METHOD M_Init : BOOL
VAR_INPUT
END_VAR
END_METHOD

METHOD ParseStateToString : STRING
VAR_INPUT
END_VAR
END_METHOD

METHOD GenerateErrorMsg : STRING
VAR_INPUT
	errorType	: STRING;
//	strState	: STRING;
	iState		: INT;
	errorMsg	: STRING;
END_VAR
END_METHOD

METHOD M_Log : STRING
VAR_INPUT
	eLogType	: E_ServerityLevelType;
	sTextLog	: STRING;
END_VAR
END_METHOD

END_INTERFACE

// MyPackML/Application/PackML/PackML/Machine State/PML_StateMachine
//can be bypass the state which is disable according to the configuration of eMode
//example:if disable clearing and resetting,when it command=clear/reset it will bybass M_Clearing and M_Stopped
//output estate according to eCommand ,then the subunit call the corresponding method according to the estate
FUNCTION_BLOCK PML_StateMachine
VAR_INPUT
	eMode				: DINT	:= E_PMLProtectedUnitMode.ePMLProtUnitMode_Production;
	eCommand			: E_PMLCommand;			
	stSubUnitInfoRef	: ST_PMLSubUnitInfoRef;	//determing machine's state according to the subUnits		
	stOptions			: ST_PMLStateMachineOptions;		
END_VAR
VAR_OUTPUT
	eState		:E_PMLState	:= ePMLState_Undefined;
	sState		:STRING;		
	bError		:BOOL;	
	nErrorID	:UDINT;	
END_VAR
VAR
	eCurrentState	: E_PMLState	:= ePMLState_Undefined;
	dwSupportedStates : DWORD := 2#11111111111111111; // Supported states
	bInit: BOOL;
END_VAR

PROPERTY _supportedStates : DWORD
GET
_supportedStates	:= dwSupportedStates;
END_GET
SET
END_SET
END_PROPERTY

// Get the next machine state without checking the supported states.
//todo:get the next machine state with checking the supported states
METHOD M_NextState : E_PMLState
VAR_INPUT
	e : E_PMLState;
END_VAR
CASE e OF
ePMLState_Stopped:
	M_NextState := ePMLState_Resetting;
ePMLState_Resetting:
	M_NextState := ePMLState_Idle;
ePMLState_Idle:
	M_NextState := ePMLState_Starting;
ePMLState_Starting:
	M_NextState := ePMLState_Execute;
ePMLState_Execute://
	M_NextState := ePMLState_Undefined;
ePMLState_Holding:
	M_NextState := ePMLState_Held;
ePMLState_Held:
	M_NextState := ePMLState_Unholding;
ePMLState_Unholding:
	M_NextState := ePMLState_Execute;
ePMLState_Suspending:
	M_NextState := ePMLState_Suspended;
ePMLState_Suspended:
	M_NextState := ePMLState_Unsuspending;
ePMLState_Unsuspending:
	M_NextState := ePMLState_Execute;
ePMLState_Completing:
	M_NextState := ePMLState_Complete;
ePMLState_Complete:
	M_NextState := ePMLState_Resetting;
ePMLState_Stopping:	
	M_NextState := ePMLState_Stopped;
ePMLState_Aborting:
	M_NextState := ePMLState_Aborted;
ePMLState_Aborted:
	M_NextState := ePMLState_Clearing;
ePMLState_Clearing:
	M_NextState := ePMLState_Stopped;
END_CASE
END_METHOD

// This method should be called by the program if an action has been finished.
//if not 
METHOD M_StateComplete : BOOL
VAR_INPUT
END_VAR
CASE eState OF
	ePMLState_Undefined:
		M_StateComplete	:= FALSE;
	ePMLState_Clearing:
		IF (TO_DWORD(M_NextState(eState)) AND _supportedStates) = 0 THEN//disable clearing
			M_StateComplete := FALSE;
			RETURN;
		END_IF	
		eState := M_NextState(eState);
		M_StateComplete := TRUE;
	ePMLState_Starting:
	//
	ePMLState_Stopping:	
	//
	ePMLState_Aborting:
	//
	ePMLState_Holding:
	//
	ePMLState_Unholding:
	//
	ePMLState_Suspending:
	//
	ePMLState_Unsuspending:
	//
	ePMLState_Resetting:
	//
	ePMLState_Completing:
	//
	
	
	
	ePMLState_Complete:
	//
	ePMLState_Stopped:
	//	
	ePMLState_Idle:
	//
	ePMLState_Suspended:
	//
	ePMLState_Execute:
	//
	ePMLState_Aborted:
	//
	ePMLState_Held:
	//
END_CASE
END_METHOD

END_FUNCTION_BLOCK

// MyPackML/Application/PackML/FB_Generic
//the functionblock FB_Generick is transmitted to every machineunit
FUNCTION_BLOCK FB_Generic IMPLEMENTS I_UnitState,I_SubCallback,I_Common
VAR_INPUT
	eModeCommand			: DINT;									//Mode from superior Unit
	eCommand				: E_PMLCommand := ePMLCommand_Abort;	//Command for a new state from superior unit
END_VAR
VAR_OUTPUT
	eMode					: DINT;									//Actual mode of the Unit
	eState					: E_PMLState (*:= ePMLState_Aborted*) ;	//Actual state of the Unit
	
	bUndefinedDone			: BOOL;									//When the SPS is started, the first state is Undefiend. bUndefined is TRUE, when the method Undefined has succesful finished
	bInvalidModeCommandOut	: BOOL;
	bChangeIntoProduction	: BOOL;
END_VAR
VAR
	fbUnitModeManager		: PML_UnitModeManager;					//The PML_UnitModeManager manage the Modechanges
	fbStateMachine 			: PML_StateMachine;						//The PML_StateMachine mangae the Statechanges
	
	nStateModeChange		: INT	:= 0;							//Variable to handle the modechange
	nLastState				: E_PMLState;							//Variable to store last state
	
	packTags				: ST_PackMLv30;
	i	: INT;
	
	ton_timeout			: TON;
	iStateTemp			: INT;	
	
	rTrig_electricalError	:ARRAY[0..10] OF R_TRIG;
	alarm_temp		: ST_Alarm;
	subscribed	: BOOL	:= FALSE;
	subData		: PubSubData;
	
	strState	: STRING;
	sComponent_name			: STRING;
	iComponetID				: INT;	
	infoLevel	: E_ServerityLevelType;//should be set to high level after debug
END_VAR

M_mapping();
CASE nStateModeChange OF
0:
	//Waiting for user request
	bChangeIntoProduction:= FALSE;
	IF  GVL.bButtonProductionReq AND (GVL.PackTags.Command.UnitMode = ePMLProtUnitMode_Production) AND (GVL.PackTags.Status.UnitModeCurrent = ePMLProtUnitMode_Invalid) THEN
			nStateModeChange	:= 1;
	ELSIF  GVL.PackTags.Command.UnitModeChangeRequest AND (GVL.PackTags.Command.UnitMode <> ePMLProtUnitMode_Production) THEN
			nStateModeChange	:= 1;
	ELSIF  GVL.bButtonProductionReq AND (GVL.PackTags.Command.UnitMode = ePMLProtUnitMode_Production) AND (GVL.PackTags.Status.UnitModeCurrent <> ePMLProtUnitMode_Production) THEN
			nStateModeChange	:= 3;
	END_IF
1:
	//Starting UnitModeManager 
	fbUnitModeManager.bExecute				:= TRUE;
	fbUnitModeManager.eModeCommand			:= eModeCommand;
	GVL.PackTags.Status.UnitModeChangeInProcess	:= TRUE;

	IF fbUnitModeManager.bDone THEN
		fbUnitModeManager.bExecute	:= FALSE;
		bInvalidModeCommandOut		:= FALSE;
		nStateModeChange			:= 0;
		bChangeIntoProduction		:= FALSE;
		GVL.PackTags.Status.UnitModeChangeInProcess	:= FALSE;
	ELSIF fbUnitModeManager.bError THEN
		bInvalidModeCommandOut		:= TRUE;
		fbUnitModeManager.bExecute	:= FALSE;
		nLastState					:= GVL.packTags.Status.StateCurrent;
		nStateModeChange			:= 2;
		bChangeIntoProduction		:= FALSE;
		GVL.PackTags.Status.UnitModeChangeInProcess	:= FALSE;
	END_IF
2:
	//ErrorHanddling
	IF  GVL.PackTags.Command.UnitModeChangeRequest THEN
		nStateModeChange:=0;
		bInvalidModeCommandOut		:= FALSE;
	ELSIF nLastState<> GVL.PackTags.Status.StateCurrent THEN
		bInvalidModeCommandOut		:= FALSE;
	END_IF
	
3:
	//state to check, if command 'Porduction' is valid
	IF (GVL.PackTags.Status.StateCurrent = ePMLState_Aborted OR GVL.PackTags.Status.StateCurrent = ePMLState_Stopped OR GVL.PackTags.Status.StateCurrent = ePMLState_Idle) THEN
		bChangeIntoProduction		:= TRUE;
		IF  GVL.stChangeIntoProduction.bYes OR GVL.stChangeIntoProduction.bYesReset THEN
			nStateModeChange			:= 1;		
		ELSIF GVL.stChangeIntoProduction.bNo THEN
			nStateModeChange			:= 0;
		END_IF
	ELSE
		nStateModeChange:= 2;
		bInvalidModeCommandOut		:= TRUE;
		nLastState					:= GVL.PackTags.Status.StateCurrent;
	END_IF
END_CASE


fbUnitModeManager(									
	eState			:= eState,
	eModeStatus		=> eMode,
	bDone			=> ,
	bError			=> ,
	nErrorId		=> );


IF fbUnitModeManager.eModeStatus <>  0 THEN
	//Calling the StateMachine, when there is a valid Mode
	fbStateMachine(
		eMode				:= eMode, 				
		eCommand			:= eCommand,			
		stSubUnitInfoRef	:= ,
		stOptions			:= , 
		eState				=> eState, 				
		bError				=> , 
		nErrorID			=> );
END_IF

//One of the methods is executing  by the actual state
CASE eState OF
	ePMLState_Undefined:
		M_Undefined();
	ePMLState_Clearing:
		M_Clearing();
	ePMLState_Stopped:
		M_Stopped();
	ePMLState_Starting:
		M_Starting();
	ePMLState_Idle:
		M_Idle();
	ePMLState_Suspended:
		M_Suspended();
	ePMLState_Execute:
		M_Execute();
	ePMLState_Stopping:
		M_Stopping();
	ePMLState_Aborting:
		M_Aborting();
	ePMLState_Aborted:
		M_Aborted();
	ePMLState_Holding:
		M_Holding();
	ePMLState_Held:
		M_Held();
	ePMLState_Unholding:
		M_Unholding();
	ePMLState_Suspending:
		M_Suspending();
	ePMLState_Unsuspending:
		M_Unsuspending();
	ePMLState_Resetting:
		M_Resetting();
	ePMLState_Completing:
		M_Completing();
	ePMLState_Complete:
		M_Complete();
END_CASE

{attribute 'object_name' := 'M_Clearing'}
METHOD M_Clearing
M_StateComplete();
END_METHOD

METHOD M_Init : BOOL
VAR_INPUT
END_VAR
END_METHOD

{attribute 'object_name' := 'M_Complete'}
METHOD M_Complete
END_METHOD

{attribute 'object_name' := 'M_Suspended'}
METHOD M_Suspended
END_METHOD

METHOD ParseStateToString : STRING
VAR_INPUT
END_VAR
END_METHOD

{attribute 'object_name' := 'M_Idle'}
METHOD M_Idle
END_METHOD

(*
M_Log method :
*)
METHOD M_Log : STRING
VAR_INPUT
	eLogType	: E_ServerityLevelType;
	sTextLog	: STRING;	
END_VAR
IF eLogType <= infoLevel THEN
//
END_IF
END_METHOD

{attribute 'object_name' := 'M_Held'}
METHOD M_Held
END_METHOD

{attribute 'object_name' := 'M_Aborted'}
METHOD M_Aborted
END_METHOD

(*
GenerateErrorMsg method:generate the error message according to the inputs
generate example:'{M9906} fb_sample DETECTION time out for T#3s.'
errorType:
		'M':mechanical error
		'E':electrical error
		'S':safety error
iState:state of state machine
errorMsg:descirbe the error
sComponent_name:defined in every componet
iComponetID:defined in every componet
strState:parseStateToString() to get the strState in ervery component
sTimeout_setting:defined in every componet
*)
METHOD GenerateErrorMsg : STRING
VAR_INPUT
	errorType	: STRING;
	iState		: INT;
	errorMsg	: STRING;	
END_VAR
VAR
	errorID	: INT;
END_VAR
GenerateErrorMsg	:= '';
GenerateErrorMsg	:= CONCAT('{',errorType);
IF iComponetID<10 THEN
	errorID	:= iComponetID*1000+iState;
ELSE
	errorID	:= iComponetID*100+iState;
END_IF
GenerateErrorMsg	:= CONCAT(GenerateErrorMsg,INT_TO_STRING(errorID));
GenerateErrorMsg	:= CONCAT(GenerateErrorMsg,'} ');
GenerateErrorMsg	:= CONCAT(GenerateErrorMsg,sComponent_name);
GenerateErrorMsg	:= CONCAT(GenerateErrorMsg,' ');
GenerateErrorMsg	:= CONCAT(GenerateErrorMsg,strState);
GenerateErrorMsg	:= CONCAT(GenerateErrorMsg,' ');
GenerateErrorMsg	:= CONCAT(GenerateErrorMsg,errorMsg);
IF errorMsg='time out' THEN
	GenerateErrorMsg	:= CONCAT(GenerateErrorMsg,' ');
	GenerateErrorMsg	:= CONCAT(GenerateErrorMsg,'for ');
	GenerateErrorMsg	:= CONCAT(GenerateErrorMsg,TIME_TO_STRING(ton_timeout.PT));//timeout setting
	GenerateErrorMsg	:= CONCAT(GenerateErrorMsg,'.');
END_IF
END_METHOD

{attribute 'object_name' := 'M_Completing'}
METHOD M_Completing
M_StateComplete();
END_METHOD

{attribute 'object_name' := 'M_Execute'}
METHOD M_Execute

M_StateComplete();
END_METHOD

{attribute 'object_name' := 'M_Stopped'}
METHOD M_Stopped
END_METHOD

(*
Description: 
the callback that will be invoked when there is a publish for what the subscriber was subscribed to.
*)
METHOD Callback
VAR_INPUT
	data : PubSubData;
END_VAR
END_METHOD

{attribute 'object_name' := 'M_Unsuspending'}
METHOD M_Unsuspending
VAR_INPUT
END_VAR
M_StateComplete();
END_METHOD

{attribute 'object_name' := 'M_Starting'}
METHOD M_Starting
M_StateComplete();
END_METHOD

{attribute 'object_name' := 'M_Holding'}
METHOD M_Holding
M_StateComplete();
END_METHOD

{attribute 'object_name' := 'M_Suspending'}
METHOD M_Suspending
VAR_INPUT
END_VAR
M_StateComplete();
END_METHOD

METHOD M_CheckError : BOOL
VAR_INPUT
END_VAR

VAR
	Trigger: INT;
END_VAR
M_CheckError	:= FALSE;

FOR i:=1 TO G_PML.MaxAlarms DO
	IF THIS^.PackTags.Admin.Alarm[i].Trigger THEN
		M_CheckError	:= TRUE;
	END_IF
END_FOR
END_METHOD

{attribute 'object_name' := 'M_Resetting'}
METHOD M_Resetting
M_StateComplete();
END_METHOD

{attribute 'object_name' := 'M_StateComplete'}
METHOD M_StateComplete
//the actual state is completed
fbStateMachine.M_StateComplete();
END_METHOD

{attribute 'object_name' := 'M_Aborting'}
METHOD M_Aborting
M_StateComplete();
END_METHOD

{attribute 'object_name' := 'M_Stopping'}
METHOD M_Stopping
M_StateComplete();
END_METHOD

{attribute 'object_name' := 'M_Unholding'}
METHOD M_Unholding
VAR_INPUT
END_VAR
M_StateComplete();
END_METHOD

METHOD M_mapping : BOOL
VAR_INPUT
END_VAR
alarm_temp.DateTime	:=GVL.packTags.Admin.PlcDateTime;
END_METHOD

{attribute 'object_name' := 'M_Undefined'}
METHOD M_Undefined
END_METHOD

END_FUNCTION_BLOCK

// MyPackML/Application/PackML/PackML/Machine State/PML_UnitModeManager
//if estate is enable to switch mode
FUNCTION_BLOCK PML_UnitModeManager
VAR_INPUT
	bExecute		: BOOL;				
	eModeCommand	: DINT;				
	eState			: E_PMLState;	//for decide if mode can be change,if can,change and done,if not,error with errorid	
END_VAR
VAR_OUTPUT
	eModeStatus	: DINT;				
	sModeStatus	: STRING;				
	bDone		: BOOL;				
	bError		: BOOL;				
	nErrorId	: UDINT;
END_VAR
VAR
END_VAR

// Switch to an other unit mode and check the permission.
// Returns true if switching is allowed, returns false if switching is forbidden.
METHOD M_SwitchUnitMode : BOOL
VAR_INPUT
	sModeName: STRING; // Name of the unit mode to switch
END_VAR
END_METHOD

// Registers an unit mode
METHOD M_Register : BOOL
VAR_INPUT
	
END_VAR
END_METHOD

END_FUNCTION_BLOCK

// MyPackML/Application/PackML/FB_Sample
FUNCTION_BLOCK FB_Sample EXTENDS FB_Generic
VAR_INPUT
END_VAR
VAR_OUTPUT
END_VAR
VAR
	lamp			: BOOL;	
	eStates			: E_SampleStates := E_SampleStates.IDLE;;
	eStateTemp		: E_SampleStates := E_SampleStates.IDLE;
	
END_VAR

SUPER^();
IF NOT subscribed THEN
	GVL.PubSubService.Subscribe(E_Topics.SAMPLE_SUBSCRRIBE_1,THIS^);
	GVL.PubSubService.Subscribe(E_Topics.SAMPLE_SUBSCRRIBE_2,THIS^);
	GVL.PubSubService.Subscribe(E_Topics.SAMPLE_SUBSCRRIBE_3,THIS^);
END_IF
subscribed	:= TRUE;


sComponent_name		:= 'fb_sample';
iComponetID			:= 99;
strState	:= ParseStateToString();
infoLevel	:= E_ServerityLevelType.WARNING;

(*
Description: 
the callback that will be invoked when there is a publish for what the subscriber was subscribed to.
*)
METHOD Callback
VAR_INPUT
	data : PubSubData;
END_VAR
CASE data.Topic OF
	E_Topics.SAMPLE_SUBSCRRIBE_1:
		//ADSLOGSTR(msgCtrlMask:= ADSLOG_MSGTYPE_LOG,msgFmtStr:='get data from publish 1',strArg:='');
	E_Topics.SAMPLE_SUBSCRRIBE_2:
		//ADSLOGSTR(msgCtrlMask:= ADSLOG_MSGTYPE_LOG,msgFmtStr:='get data from publish 2',strArg:='');
	E_Topics.SAMPLE_SUBSCRRIBE_3:
		//ADSLOGSTR(msgCtrlMask:= ADSLOG_MSGTYPE_LOG,msgFmtStr:='get data from publish 3',strArg:='');		
END_CASE
END_METHOD

{attribute 'object_name' := 'M_Completing'}
METHOD M_Completing
CASE fbUnitModeManager.eModeStatus OF
	ePMLProtUnitMode_Production:
		;
END_CASE
END_METHOD

{attribute 'object_name' := 'M_Resetting'}
METHOD M_Resetting
CASE fbUnitModeManager.eModeStatus OF
	ePMLProtUnitMode_Production:		//Production, Mantainance, Manual
		lamp	:= FALSE;
		eStates :=E_SampleStates.IDLE;
		M_StateComplete();
	
	ePMLProtUnitMode_Maintenance, ePMLProtUnitMode_Manual, ePMLUnitMode_Service:
		M_StateComplete();
END_CASE
END_METHOD

METHOD ParseStateToString : STRING
VAR_INPUT
END_VAR
CASE THIS^.eStates OF
	E_SampleStates.IDLE:
		ParseStateToString	:='IDLE';
	E_SampleStates.INIT:
		ParseStateToString	:='INIT';
	E_SampleStates.CHECK:
		ParseStateToString	:='CHECK';
	E_SampleStates.DETECTION:	
		ParseStateToString	:='DETECTION';
	E_SampleStates.LAMP_ON:
		ParseStateToString	:='LAMP_ON';
	E_SampleStates.LAMP_OFF:
		ParseStateToString	:='LAMP_OFF';
	E_SampleStates.WAIT:
		ParseStateToString	:='WAIT';
	E_SampleStates.WAIT_ON:
		ParseStateToString	:='WAIT_ON';
	E_SampleStates.WAIT_OFF:
		ParseStateToString	:='WAIT_OFF';
	E_SampleStates.DONE:	
		ParseStateToString	:='DONE';
	E_SampleStates.ERROR:
		ParseStateToString	:='ERROR';
	ELSE
		ParseStateToString	:='UNKNOW STATE';
END_CASE
END_METHOD

{attribute 'object_name' := 'M_Stopping'}
METHOD M_Stopping
CASE fbUnitModeManager.eModeStatus OF
	ePMLProtUnitMode_Production, ePMLProtUnitMode_Manual:
				//////////////////////////////////////////////////////////timeout//////////////////////////////////////////	
		iStateTemp	:= eStateTemp;
		ton_timeout();
		IF eStateTemp=eStates THEN
			ton_timeout.IN	:=TRUE;
		ELSE
			ton_timeout.IN	:=FALSE;
			eStateTemp	:= eStates;	
		END_IF
		IF ton_timeout.Q THEN	
			ton_timeout.IN	:=FALSE;
			CASE eStates OF		
				E_SampleStates.IDLE:						
					;
				E_SampleStates.INIT:
					;
				E_SampleStates.WAIT_ON:
					;
				E_SampleStates.WAIT_OFF:
					;			
				E_SampleStates.ERROR:	
					alarm_temp.Message	:= 'Sample in error state';
				ELSE
					alarm_temp.Message	:= 'UNKNOWN STATES in Sample module';
			END_CASE
			IF eStates<>E_SampleStates.IDLE AND eStates<>E_SampleStates.WAIT_ON AND eStates<>E_SampleStates.WAIT_OFF THEN
				GVL.pml_adminAlarm.M_SetAlarm(stAdmin:=GVL.PackTags.Admin,stAlarm:=alarm_temp);
			END_IF
		END_IF
		
		CASE eStates OF 
				E_SampleStates.IDLE:						
					eStates	:= E_SampleStates.INIT;				
				E_SampleStates.INIT:
					ton_timeout.PT	:= T#1S;
					eStates	:= E_SampleStates.WAIT_ON; 
				E_SampleStates.WAIT_ON:
					lamp	:= TRUE;
					IF ton_timeout.Q THEN
						eStates	:= E_SampleStates.WAIT_OFF;
					END_IF
				E_SampleStates.WAIT_OFF:
					lamp	:= FALSE;
					IF ton_timeout.Q THEN
						eStates	:= E_SampleStates.IDLE;
						M_StateComplete();	
					END_IF
				E_SampleStates.ERROR:
					;
			END_CASE			
	ePMLProtUnitMode_Maintenance, ePMLUnitMode_Service:
		M_StateComplete();	
			//not defined
END_CASE
END_METHOD

{attribute 'object_name' := 'M_Holding'}
METHOD M_Holding
CASE fbUnitModeManager.eModeStatus OF
	ePMLProtUnitMode_Production:		//Mode Production
		//Finisch the actual seperationstep	
		

	ePMLProtUnitMode_Maintenance:
		M_StateComplete();
END_CASE
END_METHOD

{attribute 'object_name' := 'M_Starting'}
METHOD M_Starting
CASE fbUnitModeManager.eModeStatus OF
	ePMLProtUnitMode_Production:		//Production, Mantainance, Manual
		
		M_StateComplete();
	ePMLProtUnitMode_Maintenance, ePMLProtUnitMode_Manual, ePMLUnitMode_Service:
		M_StateComplete();
END_CASE
END_METHOD

METHOD M_agingTest : BOOL
VAR_INPUT
	
END_VAR
END_METHOD

{attribute 'object_name' := 'M_Execute'}
METHOD M_Execute

CASE fbUnitModeManager.eModeStatus OF
	ePMLProtUnitMode_Production:		//Mode Production
		//////////////////////////////////////////////////////////timeout//////////////////////////////////////////	
		iStateTemp	:= eStateTemp;
		ton_timeout();
		IF eStateTemp=eStates THEN
			ton_timeout.IN	:=TRUE;
		ELSE
			ton_timeout.IN	:=FALSE;
			eStateTemp	:= eStates;	
			M_Log(eLogType:=E_ServerityLevelType.INFO,sTextLog:='');
			IF ton_timeout.Q THEN
				RETURN;
			END_IF
		END_IF
		IF ton_timeout.Q THEN	
			ton_timeout.IN	:=FALSE;
			CASE eStates OF	
				E_SampleStates.ERROR:	
					alarm_temp.Message	:= GenerateErrorMsg(errorType:='M',iState := iStateTemp,errorMsg:='in error state.');
				ELSE
				alarm_temp.Message	:= GenerateErrorMsg(errorType:='M',iState := iStateTemp,errorMsg:='time out');
			END_CASE
			
//			CASE eStates OF		
//				E_SampleStates.IDLE:						
//					;
//				E_SampleStates.INIT:
//					;
//				E_SampleStates.WAIT_ON:
//					;
//				E_SampleStates.WAIT_OFF:
//					;			
//				E_SampleStates.ERROR:	
//					alarm_temp.Message	:= 'Sample in error state';
//				ELSE
//					alarm_temp.Message	:= 'UNKNOWN STATES in Sample module';
//			END_CASE
			IF eStates<>E_SampleStates.IDLE AND eStates<>E_SampleStates.WAIT_ON AND eStates<>E_SampleStates.WAIT_OFF THEN
				GVL.pml_adminAlarm.M_SetAlarm(stAdmin:=GVL.PackTags.Admin,stAlarm:=alarm_temp);
			END_IF
		END_IF
		
		CASE eStates OF 
				E_SampleStates.IDLE:
					ton_timeout.PT	:= T#1MS;						
					eStates	:= E_SampleStates.INIT;				
				E_SampleStates.INIT:
					ton_timeout.PT	:= T#1S;
					eStates	:= E_SampleStates.WAIT_ON; 
				E_SampleStates.DETECTION:
					ton_timeout.PT	:= T#3S;
				E_SampleStates.WAIT:
					ton_timeout.PT	:= T#200MS;					
				E_SampleStates.WAIT_ON:
					lamp	:= TRUE;
					IF ton_timeout.Q THEN
						eStates	:= E_SampleStates.WAIT_OFF;
					END_IF
				E_SampleStates.WAIT_OFF:
					lamp	:= FALSE;
					IF ton_timeout.Q THEN
						eStates	:= E_SampleStates.IDLE;
					END_IF
				E_SampleStates.ERROR:
					;
			END_CASE
		
		
	ePMLProtUnitMode_Maintenance, ePMLUnitMode_Service:		
		//
		
	ePMLProtUnitMode_Manual:		//Manaul

END_CASE
END_METHOD

{attribute 'object_name' := 'M_Undefined'}
METHOD M_Undefined

bUndefinedDone					:= TRUE;
END_METHOD

{attribute 'object_name' := 'M_Idle'}
METHOD M_Idle
// IF G_HMI.bAging_test THEN
// 	//M_agingTest();
// END_IF
END_METHOD

METHOD M_mapping : BOOL
VAR_INPUT
END_VAR
END_METHOD

{attribute 'object_name' := 'M_Aborting'}
METHOD M_Aborting
CASE fbUnitModeManager.eModeStatus OF	
	ePMLProtUnitMode_Production, ePMLProtUnitMode_Manual:		
		lamp	:= FALSE;		
		M_StateComplete();
			
	ePMLProtUnitMode_Maintenance, ePMLUnitMode_Service:
		
		M_StateComplete();
END_CASE
END_METHOD

METHOD M_Reset
VAR_INPUT
END_VAR
//Take away all commands
IF GVL.stChangeIntoProduction.bYesReset THEN
;
END_IF
END_METHOD

END_FUNCTION_BLOCK

// MyPackML/Application/PackML/PubSub/PubSubService
FUNCTION_BLOCK PubSubService IMPLEMENTS I_PubSubService
VAR_INPUT
END_VAR
VAR_OUTPUT
END_VAR

VAR
	TopicsToSubscribers : ARRAY[0..MAX_TOPICS - 1, 0..MAX_SUBSCRIBERS_PER_TOPIC - 1] OF SubscriberCell;
	subscriberCounters : ARRAY [0..MAX_TOPICS - 1] OF INT;
END_VAR

VAR CONSTANT 
	MAX_SUBSCRIBERS_PER_TOPIC : INT := 20;
	{attribute 'analysis' := '-33'}
	MAX_TOPICS : INT := E_Topics.NUMBER_OF_TOPICS;
END_VAR

METHOD Publish
VAR_INPUT
	topic	: E_Topics;
	data	: PubSubData;
END_VAR
VAR
	index : INT;
END_VAR
FOR index := 0 TO MAX_SUBSCRIBERS_PER_TOPIC -1 BY 1 DO
	IF TopicsToSubscribers[topic, index].OCCUPIED = TRUE THEN
		TopicsToSubscribers[topic, index].subscriber.Callback(data);
	END_IF
END_FOR
END_METHOD

METHOD Subscribe : INT
VAR_INPUT
	topic	: E_Topics;
	subCallback	: I_SubCallback;
END_VAR
VAR 
	index : INT;
END_VAR
Subscribe := -1;

IF  subscriberCounters[topic] >= MAX_SUBSCRIBERS_PER_TOPIC THEN
	RETURN;
END_IF

FOR index := 0 TO (MAX_SUBSCRIBERS_PER_TOPIC - 1) BY 1 DO
	IF TopicsToSubscribers[topic, index].occupied = FALSE THEN
		TopicsToSubscribers[topic, index].occupied := TRUE;
		TopicsToSubscribers[topic, index].subscriber := subCallback;
		Subscribe := index;
		subscriberCounters[topic] := subscriberCounters[topic] + 1;
		RETURN;
	END_IF
END_FOR
END_METHOD

METHOD Unsubscribe
VAR_INPUT
	topic : E_Topics;
	subscriberID	: INT;
END_VAR
IF TopicsToSubscribers[topic, subscriberID].occupied = TRUE THEN
	TopicsToSubscribers[topic, subscriberID].occupied := FALSE;
	subscriberCounters[topic] := subscriberCounters[topic] - 1; 	
END_IF
END_METHOD

END_FUNCTION_BLOCK

// MyPackML/Application/PackML/PubSub/I_PubSubService
(*
Description:
An interface to form the contract for a basic Publisher/Subscriber service.
explaination for each method is located at the method's place.
*)
INTERFACE I_PubSubService

(*
Description:
Through this method you can unsubcribe to a topic you've already subscribed beforehand.

Params: topic - the type of topic you wish to unsubscribe to
Params: subscriberID - the ID you've received from the subscribe method.
*)
METHOD Unsubscribe
VAR_INPUT
	topic : E_Topics;
	subscriberID : INT;
END_VAR
END_METHOD

(*
Description:
Through this method you can subcribe to a topic and be notified via the I_SubCallback interface.

Params: topic - the type of topic you wish to subscribe to
Params: subCallback - is a reference to subscribe who needs to implement the O_SubCallback interface.
Return: INT - this is an ID you need to keep in order to be able to use the Unsubscribe method.
		ID > 0 is a valid ID, ID = -1 meaning the you've failed to subscribe.
*)
METHOD Subscribe : INT
VAR_INPUT
	topic : E_Topics;
	subCallback :  I_SubCallback;
END_VAR
END_METHOD

(*
Description:
Through this method you can publish data to a certain topic domain

Params: topic - the type of topic you wish to publish data to.
Params: data - the data you wish to send to said topic.
*)
METHOD Publish
VAR_INPUT
	topic : E_Topics;
	data  : PubSubData;
END_VAR
END_METHOD

END_INTERFACE

// MyPackML/Application/PackML/FB_Machine
FUNCTION_BLOCK FB_Machine EXTENDS FB_Generic
VAR_INPUT

END_VAR
VAR_OUTPUT

END_VAR
VAR	

	
	stSubModuleInfo		: ARRAY [1..iSubModule] OF ST_PMLSubUnitInfo;	//Informations about the Subunits


	
	
END_VAR
VAR CONSTANT
	iSubModule	: UDINT :=1;
END_VAR

GVL.fb_sample(
	eModeCommand:= eModeCommand, 
	eCommand:= eCommand, 
	eMode=> , 
	eState=> stSubModuleInfo[iSubModule].eState, 
	bUndefinedDone=> , 
	bInvalidModeCommandOut=> , 
	bChangeIntoProduction=> );
stSubModuleInfo[iSubModule].Active		:= TRUE;

IF  GVL.fb_sample.bUndefinedDone  THEN
	bUndefinedDone := TRUE;
END_IF

//The fbStateMachine from FB_Machine gets the Information about the states and activity from the subunits
fbStateMachine.stSubUnitInfoRef.ArraySize		:= SIZEOF(stSubModuleInfo);
fbStateMachine.stSubUnitInfoRef.NoOfSubUnits	:= iSubModule;
fbStateMachine.stSubUnitInfoRef.pArray			:= ADR(stSubModuleInfo);



//Set unit information 
M_SetUnitInfo();


SUPER^();

{attribute 'object_name' := 'M_Clearing'}
METHOD M_Clearing

CASE fbUnitModeManager.eModeStatus OF
	ePMLProtUnitMode_Production:		//Production, Mantainance, Manual
		FOR i:=1 TO MaxAlarms DO
			GVL.pml_adminAlarm.M_AcknowledgeAlarm(stAdmin:=GVL.PackTags.Admin,stAlarm:=GVL.PackTags.Admin.Alarm[i]);
			GVL.pml_adminAlarm.M_ClearAlarm(stAdmin:=GVL.PackTags.Admin,stAlarm:=GVL.PackTags.Admin.Alarm[i]);
		END_FOR	
		M_StateComplete();		
// 		IF MAIN.application.safety.M_reset() THEN
// 			IF MAIN.application.safety.xError THEN
// 				eCommand	:= ePMLCommand_Abort;
// 			ELSE
// 				M_StateComplete();
// 			END_IF
// 		END_IF	
		
	
	ePMLProtUnitMode_Maintenance, ePMLProtUnitMode_Manual, ePMLUnitMode_Service:
		M_StateComplete();
END_CASE
END_METHOD

{attribute 'object_name' := 'M_Starting'}
METHOD M_Starting
CASE fbUnitModeManager.eModeStatus OF
	ePMLProtUnitMode_Production:		//Production, Mantainance, Manual
		//Resetting all Commands and Value
// 		G_HMI.bAging_test	:= FALSE;
		M_StateComplete();
	ePMLProtUnitMode_Maintenance, ePMLProtUnitMode_Manual, ePMLUnitMode_Service:
		M_StateComplete();
END_CASE
END_METHOD

METHOD M_SetUnitInfo
VAR_INPUT
END_VAR
GVL.aUnitInfo[eMachine].Name			:= 'fbMachine';
GVL.aUnitInfo[eMachine].ActMode			:= eMode;
GVL.aUnitInfo[eMachine].ActState		:= eState;

GVL.aUnitInfo[eSample].Name				:= 'fb_sample';
GVL.aUnitInfo[eSample].ActMode			:= GVL.fb_sample.eMode;
GVL.aUnitInfo[eSample].ActState			:= GVL.fb_sample.eState;
END_METHOD

{attribute 'object_name' := 'M_Resetting'}
METHOD M_Resetting
CASE fbUnitModeManager.eModeStatus OF
	ePMLProtUnitMode_Production:		//Production, Mantainance, Manual	
// 		IF MAIN.application.safety.M_reset() THEN
// 			IF MAIN.application.safety.xError THEN
// 				eCommand	:= ePMLCommand_Abort;
// 			ELSE
// 				M_StateComplete();
// 			END_IF
// 		END_IF	
		M_StateComplete();
	
	ePMLProtUnitMode_Maintenance, ePMLProtUnitMode_Manual, ePMLUnitMode_Service:
		M_StateComplete();
END_CASE
END_METHOD

END_FUNCTION_BLOCK

// MyPackML/Application/PackML/MyUnitModeManager
FUNCTION_BLOCK MyUnitModeManager
VAR_INPUT
END_VAR
VAR_OUTPUT
END_VAR
VAR
END_VAR

END_FUNCTION_BLOCK

// Device/PackMLUnitModeManager/Visualization
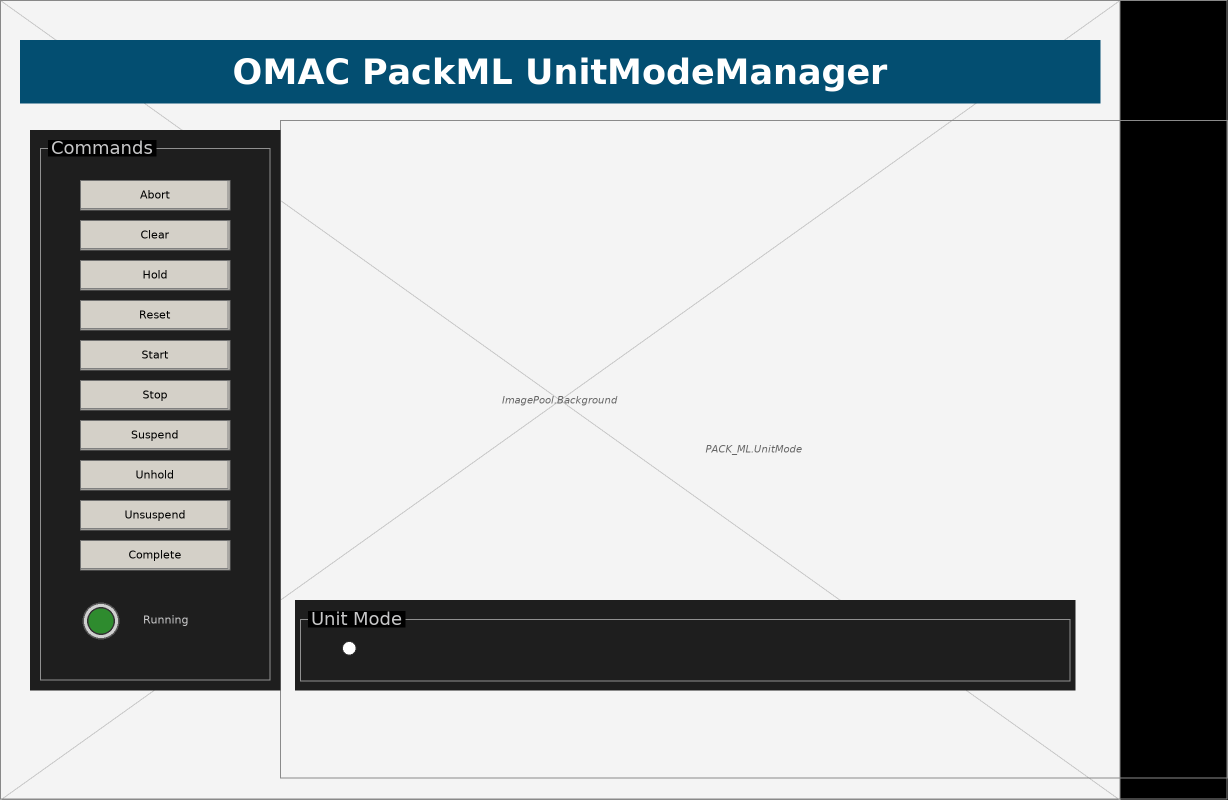
VISUALIZATION Visualization  // 1228x800
    Image (0,0 1120x800), image: ImagePool.Background
    Frame (280,120 948x658)
        shows PACK_ML.UnitMode(um := PLC_PRG.currentUnitMode)
    Rectangle (295,600 780x90)
    Rectangle (30,130 250x560)
    GroupBox (40,140 230x540), "Commands"
        Lamp1 (40,460 42x42), variable: PLC_PRG.xSimulate, style: Lamp-Lamp1-Green
        Label (100,465 57x30), "Running"
        Button (40,40 150x30), "Abort"
            tap PLC_PRG.xAbort
        Button (40,80 150x30), "Clear"
            tap PLC_PRG.xClear
        Button (40,120 150x30), "Hold"
            tap PLC_PRG.xHold
        Button (40,160 150x30), "Reset"
            tap PLC_PRG.xReset
        Button (40,200 150x30), "Start"
            tap PLC_PRG.xStart
        Button (40,240 150x30), "Stop"
            tap PLC_PRG.xStop
        Button (40,280 150x30), "Suspend"
            tap PLC_PRG.xSuspend
        Button (40,320 150x30), "Unhold"
            tap PLC_PRG.xUnHold
        Button (40,360 150x30), "Unsuspend"
            tap PLC_PRG.xUnSuspend
        Button (40,400 150x30), "Complete"
            tap PLC_PRG.xActingStateComplete
    GroupBox (300,611 770x70), "Unit Mode"
        RadioButton (40,20 700x34), variable: PLC_PRG.iSelectedUnitMode
            Areas[0]: Text=Production
            Areas[1]: Text=Semi Auto Production
            Areas[2]: Text=Setup
    Rectangle (20,40 1080x63), "OMAC PackML UnitModeManager"
END_VISUALIZATION

// Device2/PackMLAxisControl/Visualization
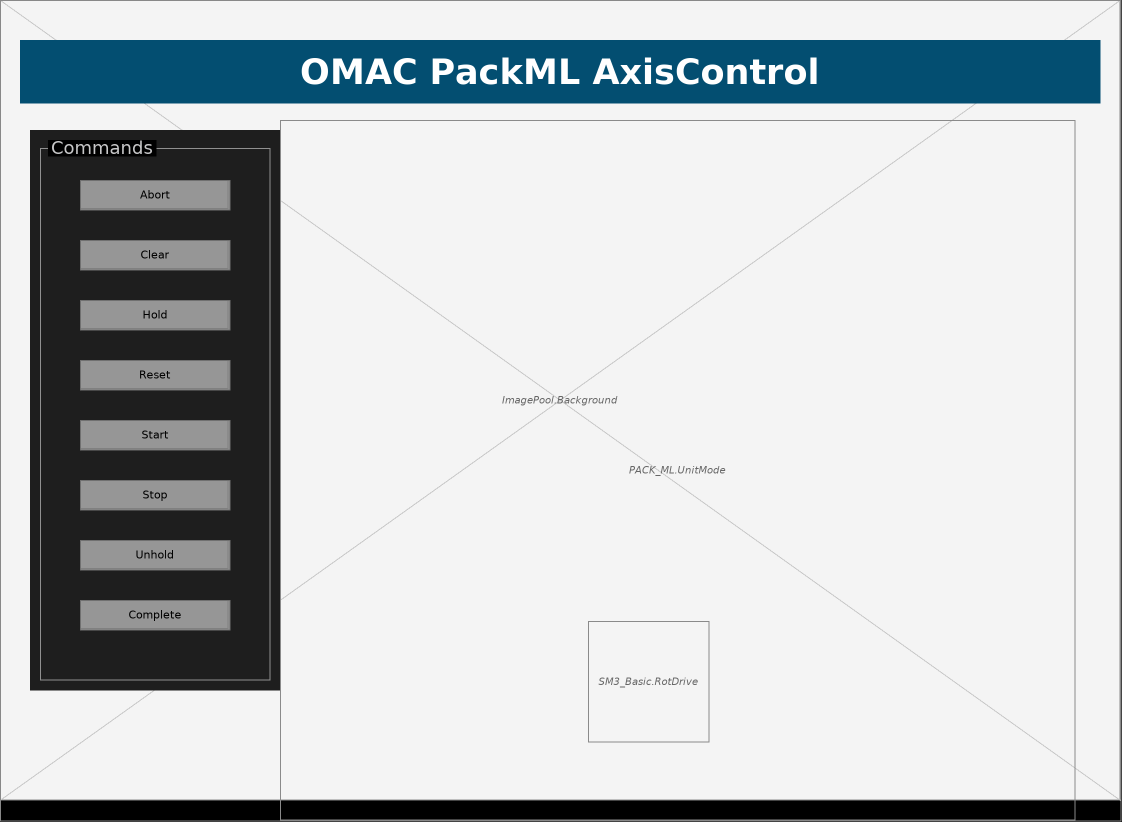
VISUALIZATION Visualization  // 1122x822
    Image (0,0 1120x800), image: ImagePool.Background
    Rectangle (30,130 250x560)
    GroupBox (40,140 230x540), "Commands"
        Button (40,40 150x30), "Abort"
            tap PLC_PRG.xAbort
        Button (40,100 150x30), "Clear"
            tap PLC_PRG.xClear
        Button (40,160 150x30), "Hold"
            tap PLC_PRG.xHold
        Button (40,220 150x30), "Reset"
            tap PLC_PRG.xReset
        Button (40,280 150x30), "Start"
            tap PLC_PRG.xStart
        Button (40,340 150x30), "Stop"
            tap PLC_PRG.xStop
        Button (40,400 150x30), "Unhold"
            tap PLC_PRG.xUnHold
        Button (40,460 150x30), "Complete"
            tap PLC_PRG.xActingStateComplete
    Frame (280,120 795x700)
        shows PACK_ML.UnitMode(um := PLC_PRG.ac.UM)
    Frame (588,621 121x121)
        shows SM3_Basic.RotDrive(m_Input_AXISREF := Axis)
    Rectangle (20,40 1080x63), "OMAC PackML AxisControl"
END_VISUALIZATION
